% RSLogix 500 project TON Timer.RSS, saved by version 8.30.00.16 %
PROJECT "UNTITLED"    % processor: Bul.1763 MicroLogix 1100 Series B %

PROGRAM FILES
  LAD 2   5 rungs

DATA FILES
  O0 OUTPUT  4 elements
  I1 INPUT  6 elements
  S2 STATUS  66 elements
  B3 BINARY  1 elements
  T4 TIMER  1 elements
  C5 COUNTER  1 elements
  R6 CONTROL  1 elements
  N7 INTEGER  1 elements
  F8 FLOAT  1 elements

LADDER 2
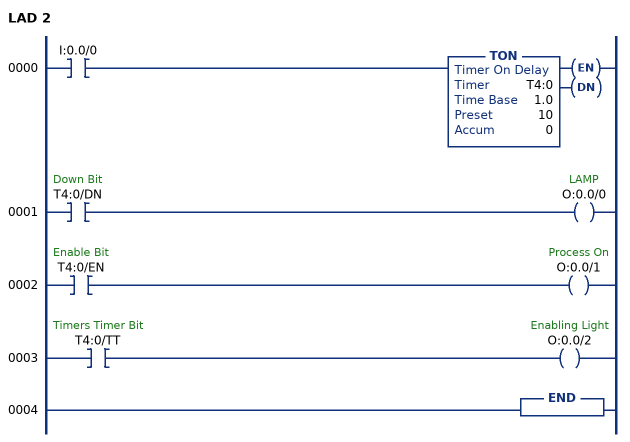
% Rung: 0 %
SOR XIC I:0.0/0 TON T4:0 1.0 10 0 EOR
% Rung: 1 %
SOR XIC T4:0/DN OTE O:0.0/0 EOR
%   T4:0/DN  "Down Bit" %
%   O:0.0/0  LAMP %
% Rung: 2 %
SOR XIC T4:0/EN OTE O:0.0/1 EOR
%   T4:0/EN  "Enable Bit" %
%   O:0.0/1  "Process On" %
% Rung: 3 %
SOR XIC T4:0/TT OTE O:0.0/2 EOR
%   T4:0/TT  "Timers Timer Bit" %
%   O:0.0/2  "Enabling Light" %
% Rung: 4 %
SOR END EOR

OTHER DOCUMENTED ADDRESSES
  I:0.0/1  "Switch1"

DATA TABLE (non-zero values as saved)
DATA T4
% .PRE .ACC %
% T4:0 % 10 0
